FUNCTION_BLOCK FB_TPD_CANopen
VAR_INPUT
	Node_address:STRING; (*CANopen node address of DCV*)
	Enable:BOOL;
	Start:BOOL;
	Reset:BOOL;
	Torque_control:BOOL;
	Speed_ref:REAL; (*Speed ref in m/s (with drive ramp)*)
	Torque_ref:REAL; (*Torque ref  in Amps for DC or as a percent of full load current for AC*)
	Nominal_speed:REAL; (*Speed in m/s at rated motor rpm*)
	Current_limit_P:REAL;
	Current_limit_N:REAL;
	Speed_P:REAL;
	Speed_I:REAL;
	Write_config:BOOL;
	Check_config:BOOL;
	Base_settings:dut_TPD32_base_settings;
	Status_word:REAL; (*DCV status word - adheres to DRIVECOM standard - same as ATV71*)
	PDO_TX1:REAL; (*DCV transmit PDO 1*)
	PDO_TX2:REAL; (*DCV transmit PDO 2*)
	PDO_TX3:REAL; (*DCV transmit PDO 3*)
END_VAR
VAR_OUTPUT
	Running:BOOL; (*Drive enabled and operational - from Control Word*)
	Fault:BOOL; (*Drive is reporting a malfunction*)
	hmi_Motor_speed:dut_hmi_Analogue; (*Motor speed in rpm*)
	hmi_Amature_current:dut_hmi_Analogue; (*Armature current as % of full load current*)
	hmi_Field_current:dut_hmi_Analogue; (*Field current as % of nominal field current*)
	hmi_Amature_voltage:dut_hmi_Analogue; (*Armature voltage in volts*)
	Mains_failure:BOOL;
	Field_failure:BOOL;
	Configuring:BOOL;
	Config_mismatch:BOOL;
	Virt_dig_in:REAL; (*DCV virtual digital inputs*)
	PDO_RX1:REAL; (*DCV receive PDO 1*)
	PDO_RX2:REAL; (*DCV receive PDO 2*)
	PDO_RX3:REAL; (*DCV receive PDO 3*)
END_VAR
VAR
	GEST1:ARRAY[1..4]OF REAL;
	Node_addm:ARRAY[0..8]OF REAL;
	Topo_address:STRING;
	Flux_current_array:ARRAY[1..2]OF REAL;
	i:REAL;
	Motor_speed:REAL;
	Amature_current:REAL;
	Amature_voltage:REAL;
	Field_current:REAL;
END_VAR
{warning 'TODO: Var Status_word was set as an INT in the original program. I have set it as a REAL as per our current structure, but should this not be a word?'}
{warning 'TODO: This function block needs to be reworked to work on our new comms'}

M_DCV_PDO();
M_DCV_config();
M_Settings();
M_DCV_analogues();

METHOD M_DCV_PDO
VAR_INPUT
END_VAR
{warning 'TODO: these comms need to be recreated as EtherCat comms I assume? The ADDM FB doesn't exist here.'}
VAR_INST // added by the converter: edge detectors and wires of the graphical bodies
    _w1 : STRING;
END_VAR
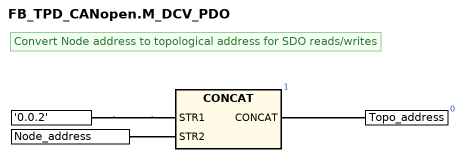
Topo_address := _w1;
// Convert Node address to topological address for SDO reads/writes
_w1 := CONCAT(STR1 := '0.0.2', STR2 := Node_address);
END_METHOD

END_FUNCTION_BLOCK

(* stored: Version 1.1.0.1, ProductVersion 3.1.4024.0
   POU FB_TPD_CANopen: Id {aba12aa0-774e-4307-bc34-d6e83193ae31}, SpecialFunc None
   Method M_DCV_PDO: Id {42f5b0e0-bb4d-4e0c-88e4-1f41f55fe8f5} *)
